FUNCTION_BLOCK FB_BPRequestor
VAR_INPUT
	stReqBP	:	ST_ReqBeamParams;
END_VAR
VAR_OUTPUT
END_VAR
VAR
	{attribute 'TcLinkTo' := 'TIIB[PMPS_IF2]^IO Outputs^ReqBP'}
	q_stReqBP	AT	%Q*	:	ST_ReqBeamParams;
END_VAR

q_stReqBP := stReqBP;

END_FUNCTION_BLOCK

(* stored: Version 1.1.0.1, ProductVersion 3.1.4022.12
   POU FB_BPRequestor: Id {7bca38cb-b015-0bee-2b8d-d1d37159090d}, SpecialFunc None *)
